// Mitsubishi GX Works2 project: 順次回路234   PLC: Q03UDV

PROGRAM MAIN
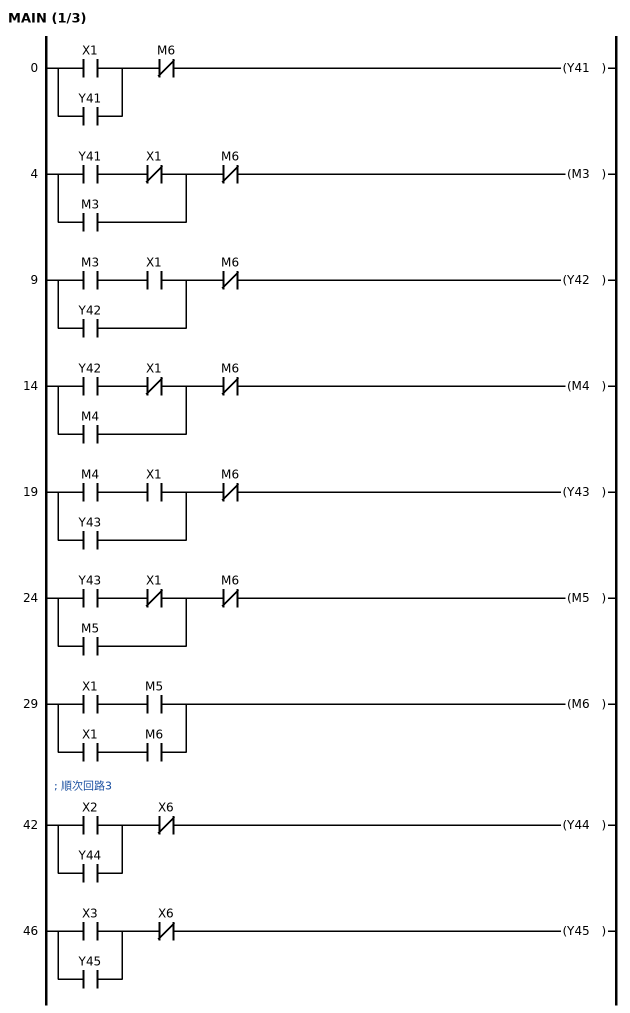
0     LD      X1
      OR      Y41
      ANI     M6
      OUT     Y41
4     LD      Y41
      ANI     X1
      OR      M3
      ANI     M6
      OUT     M3
9     LD      M3
      AND     X1
      OR      Y42
      ANI     M6
      OUT     Y42
14    LD      Y42
      ANI     X1
      OR      M4
      ANI     M6
      OUT     M4
19    LD      M4
      AND     X1
      OR      Y43
      ANI     M6
      OUT     Y43
24    LD      Y43
      ANI     X1
      OR      M5
      ANI     M6
      OUT     M5
29    LD      X1
      AND     M5
      LD      X1
      AND     M6
      ORB
      OUT     M6
; 順次回路3
42    LD      X2
      OR      Y44
      ANI     X6
      OUT     Y44
46    LD      X3
      OR      Y45
      ANI     X6
      OUT     Y45
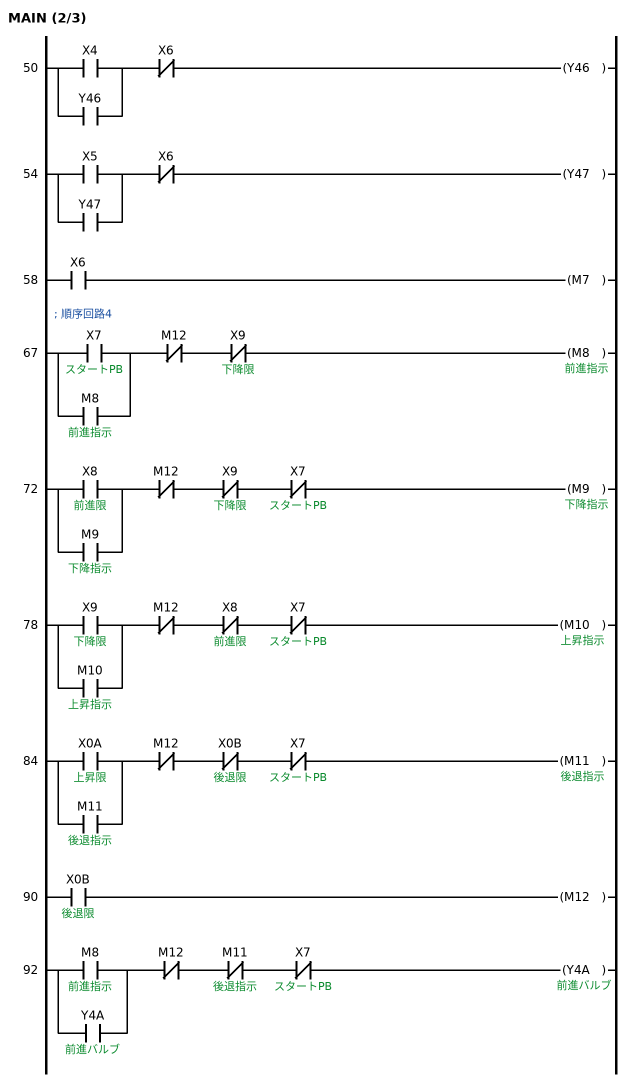
50    LD      X4
      OR      Y46
      ANI     X6
      OUT     Y46
54    LD      X5
      OR      Y47
      ANI     X6
      OUT     Y47
58    LD      X6
      OUT     M7
; 順序回路4
67    LD      X7  ; スタートPB
      OR      M8  ; 前進指示
      ANI     M12
      ANI     X9  ; 下降限
      OUT     M8  ; 前進指示
72    LD      X8  ; 前進限
      OR      M9  ; 下降指示
      ANI     M12
      ANI     X9  ; 下降限
      ANI     X7  ; スタートPB
      OUT     M9  ; 下降指示
78    LD      X9  ; 下降限
      OR      M10  ; 上昇指示
      ANI     M12
      ANI     X8  ; 前進限
      ANI     X7  ; スタートPB
      OUT     M10  ; 上昇指示
84    LD      X0A  ; 上昇限
      OR      M11  ; 後退指示
      ANI     M12
      ANI     X0B  ; 後退限
      ANI     X7  ; スタートPB
      OUT     M11  ; 後退指示
90    LD      X0B  ; 後退限
      OUT     M12
92    LD      M8  ; 前進指示
      OR      Y4A  ; 前進バルブ
      ANI     M12
      ANI     M11  ; 後退指示
      ANI     X7  ; スタートPB
      OUT     Y4A  ; 前進バルブ
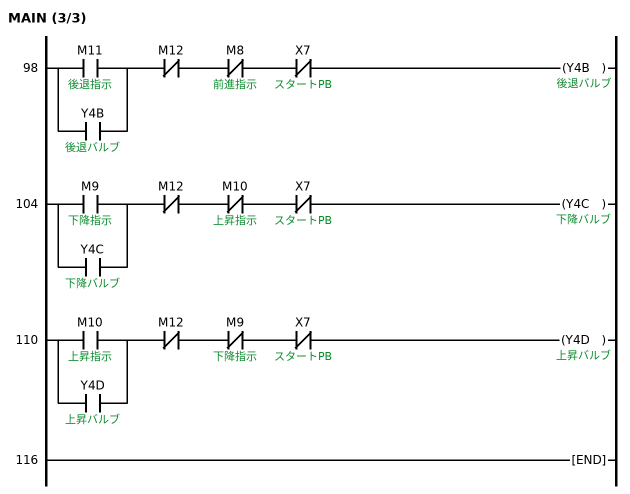
98    LD      M11  ; 後退指示
      OR      Y4B  ; 後退バルブ
      ANI     M12
      ANI     M8  ; 前進指示
      ANI     X7  ; スタートPB
      OUT     Y4B  ; 後退バルブ
104   LD      M9  ; 下降指示
      OR      Y4C  ; 下降バルブ
      ANI     M12
      ANI     M10  ; 上昇指示
      ANI     X7  ; スタートPB
      OUT     Y4C  ; 下降バルブ
110   LD      M10  ; 上昇指示
      OR      Y4D  ; 上昇バルブ
      ANI     M12
      ANI     M9  ; 下降指示
      ANI     X7  ; スタートPB
      OUT     Y4D  ; 上昇バルブ
116   END
END_PROGRAM

// device comments not shown above
Y48  ; 前進バルブ
Y49  ; 後退バルブ
